(* Logix 5000 project; controller Arrow3 vendor 1 type 14 code 235 rev 36.11; software revision 36.00; part 2 of 3 *)
(* tags used below, declared in another part *)
   b : BOOL;
   off_delay_timer : TIMER;
   on : BOOL;
   On_Delay_Timer_1 : TIMER;
   On_Delay_Timer_2 : TIMER;
   On_Delay_Timer_3 : TIMER;
   On_Delay_Timer_4 : TIMER;
   On_Delay_Timer_5 : TIMER;
   On_Delay_Timer_6 : TIMER;
   On_Delay_Timer_7 : TIMER;
   On_Delay_Timer_8 : TIMER;
   on_delay_tmr : TIMER;
   PROP_BCKPLANE_IDENT_DEVICEID_GET : MESSAGE;
   PROP_BCKPLANE_IDENT_DEVICEID_TRG_GET : BOOL;
   PROP_BCKPLANE_IDENT_DEVICENAME_GET : MESSAGE;
   PROP_BCKPLANE_IDENT_DEVICENAME_TRG_GET : BOOL;
   PROP_BCKPLANE_IDENT_DEVICETYPE_GET : MESSAGE;
   PROP_BCKPLANE_IDENT_DEVICETYPE_TRG_GET : BOOL;
   PROP_BCKPLANE_IDENT_HWREV_GET : MESSAGE;
   PROP_BCKPLANE_IDENT_HWREV_TRG_GET : BOOL;
   PROP_BCKPLANE_IDENT_SERIALNO_GET : MESSAGE;
   PROP_BCKPLANE_IDENT_SERIALNO_TRG_GET : BOOL;
   PROP_BCKPLANE_IDENT_SWPARTNO_GET : MESSAGE;
   PROP_BCKPLANE_IDENT_SWPARTNO_TRG_GET : BOOL;
   PROP_BCKPLANE_IDENT_SWREV_GET : MESSAGE;
   PROP_BCKPLANE_IDENT_SWREV_TRG_GET : BOOL;
   PROP_BCKPLANE_IDENT_VARIANTID_GET : MESSAGE;
   PROP_BCKPLANE_IDENT_VARIANTID_TRG_GET : BOOL;
   PROP_BCKPLANE_IDENT_VENDORID_GET : MESSAGE;
   PROP_BCKPLANE_IDENT_VENDORID_TRG_GET : BOOL;
   PROP_BCKPLANE_IDENT_VENDORNAME_GET : MESSAGE;
   PROP_BCKPLANE_IDENT_VENDORNAME_TRG_GET : BOOL;
   PROP_INTR_CONTROL_KD_GET : MESSAGE;
   PROP_INTR_CONTROL_KD_SET : MESSAGE;
   PROP_INTR_CONTROL_KD_TRG_GET : BOOL;
   PROP_INTR_CONTROL_KD_TRG_SET : BOOL;
   PROP_INTR_CONTROL_KI_GET : MESSAGE;
   PROP_INTR_CONTROL_KI_SET : MESSAGE;
   PROP_INTR_CONTROL_KI_TRG_GET : BOOL;
   PROP_INTR_CONTROL_KI_TRG_SET : BOOL;
   PROP_INTR_CONTROL_KP_GET : MESSAGE;
   PROP_INTR_CONTROL_KP_SET : MESSAGE;
   PROP_INTR_CONTROL_KP_TRG_GET : BOOL;
   PROP_INTR_CONTROL_KP_TRG_SET : BOOL;
   PROP_INTR_CONTROL_LCDBRIGHT_GET : MESSAGE;
   PROP_INTR_CONTROL_LCDBRIGHT_SET : MESSAGE;
   PROP_INTR_CONTROL_LCDBRIGHT_TRG_GET : BOOL;
   PROP_INTR_CONTROL_LCDBRIGHT_TRG_SET : BOOL;
   PROP_INTR_CONTROL_SPANADJST_GET : MESSAGE;
   PROP_INTR_CONTROL_SPANADJST_SET : MESSAGE;
   PROP_INTR_CONTROL_SPANADJST_TRG_GET : BOOL;
   PROP_INTR_CONTROL_SPANADJST_TRG_SET : BOOL;
   PROP_INTR_CONTROL_ZEROADJST_GET : MESSAGE;
   PROP_INTR_CONTROL_ZEROADJST_SET : MESSAGE;
   PROP_INTR_CONTROL_ZEROADJST_TRG_GET : BOOL;
   PROP_INTR_CONTROL_ZEROADJST_TRG_SET : BOOL;
   PROP_INTR_CYCLECOUNTER_GET : MESSAGE;
   PROP_INTR_CYCLECOUNTER_TRG_GET : BOOL;
   PROP_INTR_IDENT_DEVICEID_GET : MESSAGE;
   PROP_INTR_IDENT_DEVICEID_TRG_GET : BOOL;
   PROP_INTR_IDENT_DEVICENAME_GET : MESSAGE;
   PROP_INTR_IDENT_DEVICENAME_TRG_GET : BOOL;
   PROP_INTR_IDENT_DEVICETYPE_GET : MESSAGE;
   PROP_INTR_IDENT_DEVICETYPE_TRG_GET : BOOL;
   PROP_INTR_IDENT_HWREV_GET : MESSAGE;
   PROP_INTR_IDENT_HWREV_TRG_GET : BOOL;
   PROP_INTR_IDENT_SERIALNO_GET : MESSAGE;
   PROP_INTR_IDENT_SERIALNO_TRG_GET : BOOL;
   PROP_INTR_IDENT_SWPARTNO_GET : MESSAGE;
   PROP_INTR_IDENT_SWPARTNO_TRG_GET : BOOL;
   PROP_INTR_IDENT_SWREV_GET : MESSAGE;
   PROP_INTR_IDENT_SWREV_TRG_GET : BOOL;
   PROP_INTR_IDENT_VARIANTID_GET : MESSAGE;
   PROP_INTR_IDENT_VARIANTID_TRG_GET : BOOL;
   PROP_INTR_IDENT_VENDORID_GET : MESSAGE;
   PROP_INTR_IDENT_VENDORID_TRG_GET : BOOL;
   PROP_INTR_IDENT_VENDORNAME_GET : MESSAGE;
   PROP_INTR_IDENT_VENDORNAME_TRG_GET : BOOL;
   PROP_INTR_OPRHR_GET : MESSAGE;
   PROP_INTR_OPRHR_TRG_GET : BOOL;
   PROP_INTR_POST_ERRSTS_GET : MESSAGE;
   PROP_INTR_POST_ERRSTS_TRG_GET : BOOL;
   STA_ApplPresHysteresis_GET : MESSAGE;
   STA_ApplPresHysteresis_SET : MESSAGE;
   STA_ApplPresHysteresis_TRG_GET : BOOL;
   STA_ApplPresHysteresis_TRG_SET : BOOL;
   STA_Coil12HitCurHysteresis_GET : MESSAGE;
   STA_Coil12HitCurHysteresis_SET : MESSAGE;
   STA_Coil12HitCurHysteresis_TRG_GET : BOOL;
   STA_Coil12HitCurHysteresis_TRG_SET : BOOL;
   STA_Coil12HitCurrent_GET : MESSAGE;
   STA_Coil12HitCurrent_TRG_GET : BOOL;
   STA_Coil12HitPower_GET : MESSAGE;
   STA_Coil12HitPower_TRG_GET : BOOL;
   STA_Coil12HoldCurrent_GET : MESSAGE;
   STA_Coil12HoldCurrent_TRG_GET : BOOL;
   STA_Coil12HoldPower_GET : MESSAGE;
   STA_Coil12HoldPower_SET : MESSAGE;
   STA_Coil12HoldPower_TRG_GET : BOOL;
   STA_Coil12HoldPower_TRG_SET : BOOL;
   STA_Coil12HoldVolage_GET : MESSAGE;
   STA_Coil12HoldVolage_SET : MESSAGE;
   STA_Coil12HoldVolage_TRG_GET : BOOL;
   STA_Coil12HoldVolage_TRG_SET : BOOL;
   STA_Coil14HitCurHysteresis_GET : MESSAGE;
   STA_Coil14HitCurHysteresis_SET : MESSAGE;
   STA_Coil14HitCurHysteresis_TRG_GET : BOOL;
   STA_Coil14HitCurHysteresis_TRG_SET : BOOL;
   STA_Coil14HitCurrent_GET : MESSAGE;
   STA_Coil14HitCurrent_TRG_GET : BOOL;
   STA_Coil14HitPower_GET : MESSAGE;
   STA_Coil14HitPower_TRG_GET : BOOL;
   STA_Coil14HoldCurrent_GET : MESSAGE;
   STA_Coil14HoldCurrent_TRG_GET : BOOL;
   STA_Coil14HoldPower_GET : MESSAGE;
   STA_Coil14HoldPower_SET : MESSAGE;
   STA_Coil14HoldPower_TRG_GET : BOOL;
   STA_Coil14HoldPower_TRG_SET : BOOL;
   STA_Coil14HoldVolage_GET : MESSAGE;
   STA_Coil14HoldVolage_SET : MESSAGE;
   STA_Coil14HoldVolage_TRG_GET : BOOL;
   STA_Coil14HoldVolage_TRG_SET : BOOL;
   STA_DV_ERROR_STATUS_GET : MESSAGE;
   STA_DV_ERROR_STATUS_TRG_GET : BOOL;
   STA_ExhaustPresHysteresis_GET : MESSAGE;
   STA_ExhaustPresHysteresis_SET : MESSAGE;
   STA_ExhaustPresHysteresis_TRG_GET : BOOL;
   STA_ExhaustPresHysteresis_TRG_SET : BOOL;
   STA_FAULTEVNTBITS_GET : MESSAGE;
   STA_FAULTEVNTBITS_TRG_GET : BOOL;
   STA_FAULTEVNTCOUNT_GET : MESSAGE;
   STA_FAULTEVNTCOUNT_TRG_GET : BOOL;
   STA_IDENT_DEVICETYPE_GET : MESSAGE;
   STA_IDENT_DEVICETYPE_TRG_GET : BOOL;
   STA_INTR_IDENT_DEVICEID_GET : MESSAGE;
   STA_INTR_IDENT_DEVICEID_TRG_GET : BOOL;
   STA_INTR_IDENT_DEVICENAME_GET : MESSAGE;
   STA_INTR_IDENT_DEVICENAME_TRG_GET : BOOL;
   STA_INTR_IDENT_HWREV_GET : MESSAGE;
   STA_INTR_IDENT_HWREV_TRG_GET : BOOL;
   STA_INTR_IDENT_SERIALNO_GET : MESSAGE;
   STA_INTR_IDENT_SERIALNO_TRG_GET : BOOL;
   STA_INTR_IDENT_SWPARTNO_GET : MESSAGE;
   STA_INTR_IDENT_SWPARTNO_TRG_GET : BOOL;
   STA_INTR_IDENT_SWREV_GET : MESSAGE;
   STA_INTR_IDENT_SWREV_TRG_GET : BOOL;
   STA_INTR_IDENT_VARIANTID_GET : MESSAGE;
   STA_INTR_IDENT_VARIANTID_TRG_GET : BOOL;
   STA_INTR_IDENT_VENDORID_GET : MESSAGE;
   STA_INTR_IDENT_VENDORID_TRG_GET : BOOL;
   STA_INTR_IDENT_VENDORNAME_GET : MESSAGE;
   STA_INTR_IDENT_VENDORNAME_TRG_GET : BOOL;
   STA_MaxApplPressure_GET : MESSAGE;
   STA_MaxApplPressure_SET : MESSAGE;
   STA_MaxApplPressure_TRG_GET : BOOL;
   STA_MaxApplPressure_TRG_SET : BOOL;
   STA_MeasuredAuxVolt_GET : MESSAGE;
   STA_MeasuredAuxVolt_TRG_GET : BOOL;
   STA_MinApplPressure_GET : MESSAGE;
   STA_MinApplPressure_SET : MESSAGE;
   STA_MinApplPressure_TRG_GET : BOOL;
   STA_MinApplPressure_TRG_SET : BOOL;
   STA_OPERATIONTIME_HR_GET : MESSAGE;
   STA_OPERATIONTIME_HR_TRG_GET : BOOL;
   STA_OPERATIONTIME_MIN_GET : MESSAGE;
   STA_OPERATIONTIME_MIN_TRG_GET : BOOL;
   STA_Port2ApplPressCyclRating_GET : MESSAGE;
   STA_Port2ApplPressCyclRating_SET : MESSAGE;
   STA_Port2ApplPressCyclRating_TRG_GET : BOOL;
   STA_Port2ApplPressCyclRating_TRG_SET : BOOL;
   STA_Port2MesrdPressure_GET : MESSAGE;
   STA_Port2MesrdPressure_TRG_GET : BOOL;
   STA_Port2PressCycleCounter_GET : MESSAGE;
   STA_Port2PressCycleCounter_TRG_GET : BOOL;
   STA_Port2PressMonitorDly_GET : MESSAGE;
   STA_Port2PressMonitorDly_SET : MESSAGE;
   STA_Port2PressMonitorDly_TRG_GET : BOOL;
   STA_Port2PressMonitorDly_TRG_SET : BOOL;
   STA_Port4ApplPressCyclRating_GET : MESSAGE;
   STA_Port4ApplPressCyclRating_SET : MESSAGE;
   STA_Port4ApplPressCyclRating_TRG_GET : BOOL;
   STA_Port4ApplPressCyclRating_TRG_SET : BOOL;
   STA_Port4MesrdPressure_GET : MESSAGE;
   STA_Port4MesrdPressure_TRG_GET : BOOL;
   STA_Port4PressCycleCounter_GET : MESSAGE;
   STA_Port4PressCycleCounter_TRG_GET : BOOL;
   STA_Port4PressMonitorDly_GET : MESSAGE;
   STA_Port4PressMonitorDly_SET : MESSAGE;
   STA_Port4PressMonitorDly_TRG_GET : BOOL;
   STA_Port4PressMonitorDly_TRG_SET : BOOL;
   STA_PWRONTIME_HR_GET : MESSAGE;
   STA_PWRONTIME_HR_TRG_GET : BOOL;
   STA_PWRONTIME_MIN_GET : MESSAGE;
   STA_PWRONTIME_MIN_TRG_GET : BOOL;
   STA_RatedAuxVoltHyst_GET : MESSAGE;
   STA_RatedAuxVoltHyst_SET : MESSAGE;
   STA_RatedAuxVoltHyst_TRG_GET : BOOL;
   STA_RatedAuxVoltHyst_TRG_SET : BOOL;
   STA_Valve12ApplCyclRating_GET : MESSAGE;
   STA_Valve12ApplCyclRating_SET : MESSAGE;
   STA_Valve12ApplCyclRating_TRG_GET : BOOL;
   STA_Valve12ApplCyclRating_TRG_SET : BOOL;
   STA_Valve12CycleCounter_GET : MESSAGE;
   STA_Valve12CycleCounter_TRG_GET : BOOL;
   STA_Valve14ApplCyclRating_GET : MESSAGE;
   STA_Valve14ApplCyclRating_SET : MESSAGE;
   STA_Valve14ApplCyclRating_TRG_GET : BOOL;
   STA_Valve14ApplCyclRating_TRG_SET : BOOL;
   STA_Valve14CycleCounter_GET : MESSAGE;
   STA_Valve14CycleCounter_TRG_GET : BOOL;
   STA_ValveSlice12Side_GET : MESSAGE;
   STA_ValveSlice12Side_SET : MESSAGE;
   STA_ValveSlice12Side_TRG_GET : BOOL;
   STA_ValveSlice12Side_TRG_SET : BOOL;
   STA_ValveSliceFunction_GET : MESSAGE;
   STA_ValveSliceFunction_SET : MESSAGE;
   STA_ValveSliceFunction_TRG_GET : BOOL;
   STA_ValveSliceFunction_TRG_SET : BOOL;
   STA_WARNEVNTBITS_GET : MESSAGE;
   STA_WARNEVNTBITS_TRG_GET : BOOL;
   STA_WARNEVNTCOUNT_GET : MESSAGE;
   STA_WARNEVNTCOUNT_TRG_GET : BOOL;
   STA_WARNSTSBITS_GET : MESSAGE;
   STA_WARNSTSBITS_TRG_GET : BOOL;
   Station_1A : ALIAS FOR VRQx:O.Data[1].7;
   Station_1B : ALIAS FOR VRQx:O.Data[1].6;
   Station_2A : ALIAS FOR VRQx:O.Data[1].5;
   Station_2B : ALIAS FOR VRQx:O.Data[1].4;
   Station_3A : ALIAS FOR VRQx:O.Data[1].3;
   Station_3B : ALIAS FOR VRQx:O.Data[1].2;
   Station_4A : ALIAS FOR VRQx:O.Data[1].1;
   Station_4B : ALIAS FOR VRQx:O.Data[1].0;
   Station_5A : ALIAS FOR VRQx:O.Data[2].7;
   Station_5B : ALIAS FOR VRQx:O.Data[2].6;
   Station_6A : ALIAS FOR VRQx:O.Data[2].5;
   Station_6B : ALIAS FOR VRQx:O.Data[2].4;
   Station_7A : ALIAS FOR VRQx:O.Data[2].3;
   Station_7B : ALIAS FOR VRQx:O.Data[2].2;
   Station_8A : ALIAS FOR VRQx:O.Data[2].1;
   Station_8B : ALIAS FOR VRQx:O.Data[2].0;
   up_counter : COUNTER;
(* MainProgram, continued *)

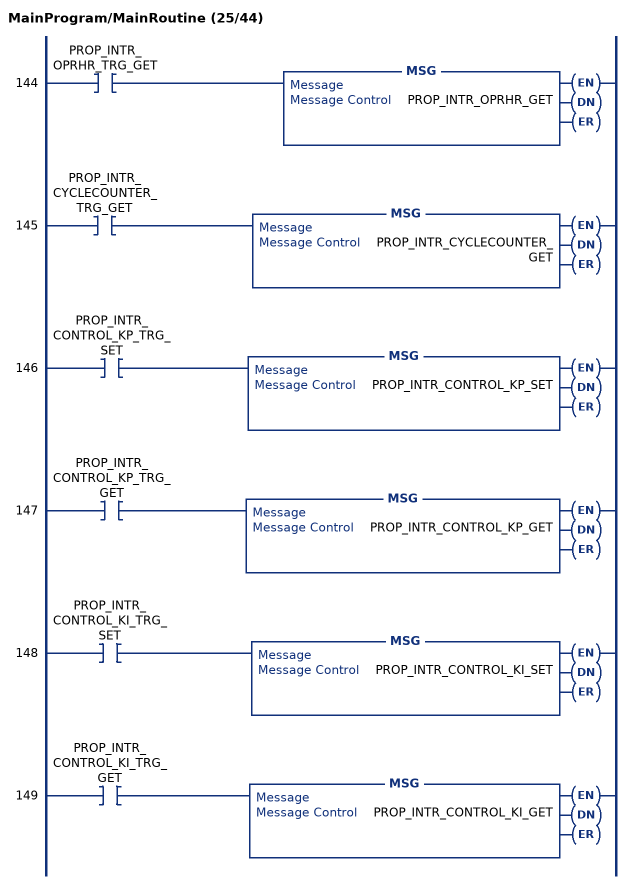
   [picture p24: MainProgram/MainRoutine rungs 144-149]
   144: XIC(PROP_INTR_OPRHR_TRG_GET)MSG(PROP_INTR_OPRHR_GET);
   145: XIC(PROP_INTR_CYCLECOUNTER_TRG_GET)MSG(PROP_INTR_CYCLECOUNTER_GET);
   146: XIC(PROP_INTR_CONTROL_KP_TRG_SET)MSG(PROP_INTR_CONTROL_KP_SET);
   147: XIC(PROP_INTR_CONTROL_KP_TRG_GET)MSG(PROP_INTR_CONTROL_KP_GET);
   148: XIC(PROP_INTR_CONTROL_KI_TRG_SET)MSG(PROP_INTR_CONTROL_KI_SET);
   149: XIC(PROP_INTR_CONTROL_KI_TRG_GET)MSG(PROP_INTR_CONTROL_KI_GET);
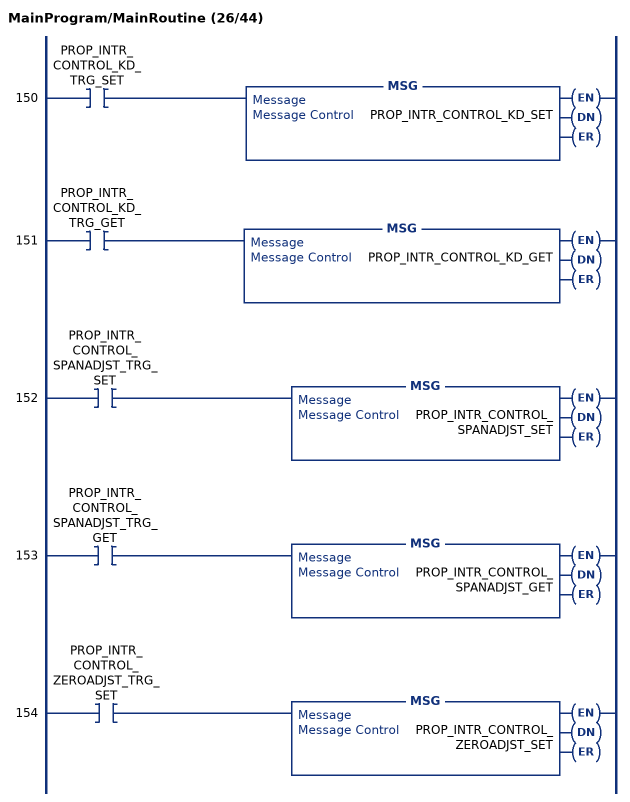
   150: XIC(PROP_INTR_CONTROL_KD_TRG_SET)MSG(PROP_INTR_CONTROL_KD_SET);
   151: XIC(PROP_INTR_CONTROL_KD_TRG_GET)MSG(PROP_INTR_CONTROL_KD_GET);
   152: XIC(PROP_INTR_CONTROL_SPANADJST_TRG_SET)MSG(PROP_INTR_CONTROL_SPANADJST_SET);
   153: XIC(PROP_INTR_CONTROL_SPANADJST_TRG_GET)MSG(PROP_INTR_CONTROL_SPANADJST_GET);
   154: XIC(PROP_INTR_CONTROL_ZEROADJST_TRG_SET)MSG(PROP_INTR_CONTROL_ZEROADJST_SET);
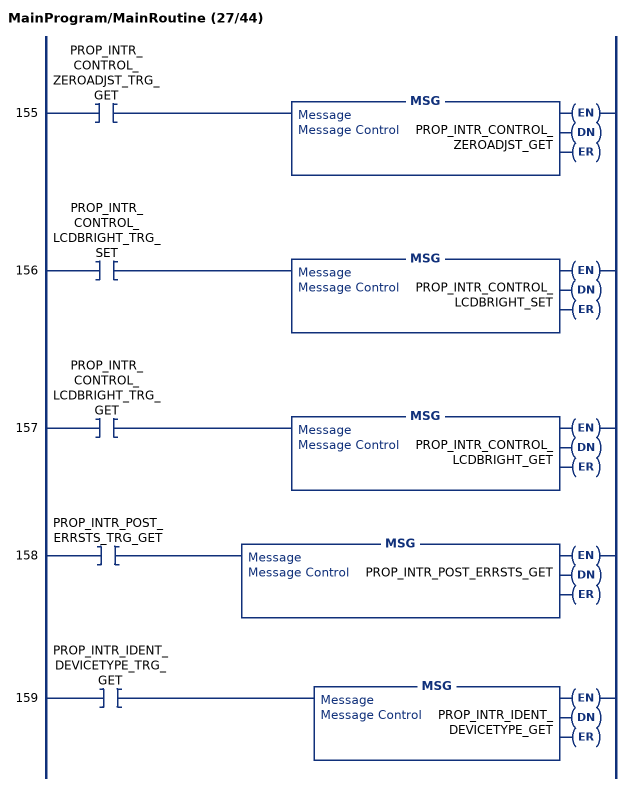
   155: XIC(PROP_INTR_CONTROL_ZEROADJST_TRG_GET)MSG(PROP_INTR_CONTROL_ZEROADJST_GET);
   156: XIC(PROP_INTR_CONTROL_LCDBRIGHT_TRG_SET)MSG(PROP_INTR_CONTROL_LCDBRIGHT_SET);
   157: XIC(PROP_INTR_CONTROL_LCDBRIGHT_TRG_GET)MSG(PROP_INTR_CONTROL_LCDBRIGHT_GET);
   158: XIC(PROP_INTR_POST_ERRSTS_TRG_GET)MSG(PROP_INTR_POST_ERRSTS_GET);
   159: XIC(PROP_INTR_IDENT_DEVICETYPE_TRG_GET)MSG(PROP_INTR_IDENT_DEVICETYPE_GET);
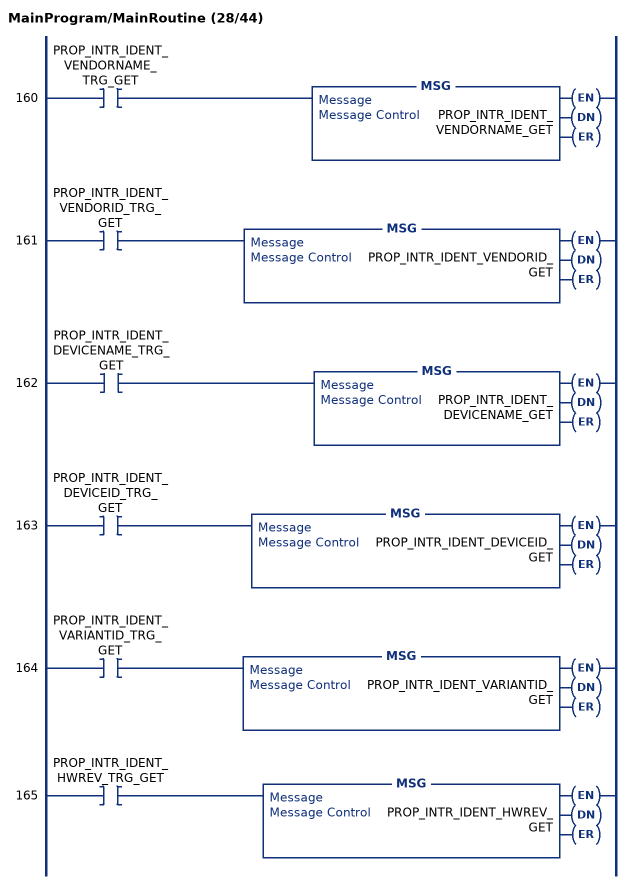
   160: XIC(PROP_INTR_IDENT_VENDORNAME_TRG_GET)MSG(PROP_INTR_IDENT_VENDORNAME_GET);
   161: XIC(PROP_INTR_IDENT_VENDORID_TRG_GET)MSG(PROP_INTR_IDENT_VENDORID_GET);
   162: XIC(PROP_INTR_IDENT_DEVICENAME_TRG_GET)MSG(PROP_INTR_IDENT_DEVICENAME_GET);
   163: XIC(PROP_INTR_IDENT_DEVICEID_TRG_GET)MSG(PROP_INTR_IDENT_DEVICEID_GET);
   164: XIC(PROP_INTR_IDENT_VARIANTID_TRG_GET)MSG(PROP_INTR_IDENT_VARIANTID_GET);
   165: XIC(PROP_INTR_IDENT_HWREV_TRG_GET)MSG(PROP_INTR_IDENT_HWREV_GET);
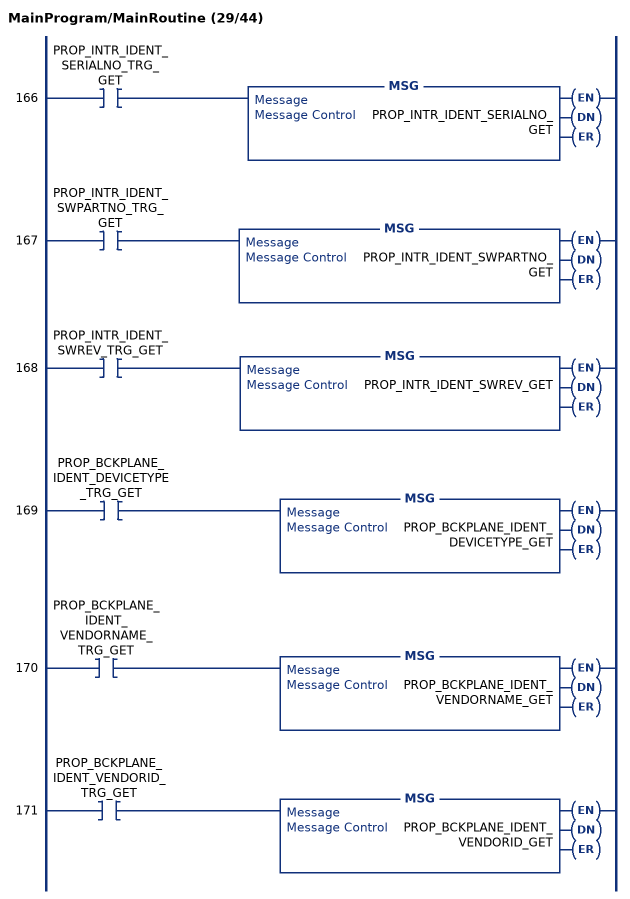
   166: XIC(PROP_INTR_IDENT_SERIALNO_TRG_GET)MSG(PROP_INTR_IDENT_SERIALNO_GET);
   167: XIC(PROP_INTR_IDENT_SWPARTNO_TRG_GET)MSG(PROP_INTR_IDENT_SWPARTNO_GET);
   168: XIC(PROP_INTR_IDENT_SWREV_TRG_GET)MSG(PROP_INTR_IDENT_SWREV_GET);
   169: XIC(PROP_BCKPLANE_IDENT_DEVICETYPE_TRG_GET)MSG(PROP_BCKPLANE_IDENT_DEVICETYPE_GET);
   170: XIC(PROP_BCKPLANE_IDENT_VENDORNAME_TRG_GET)MSG(PROP_BCKPLANE_IDENT_VENDORNAME_GET);
   171: XIC(PROP_BCKPLANE_IDENT_VENDORID_TRG_GET)MSG(PROP_BCKPLANE_IDENT_VENDORID_GET);
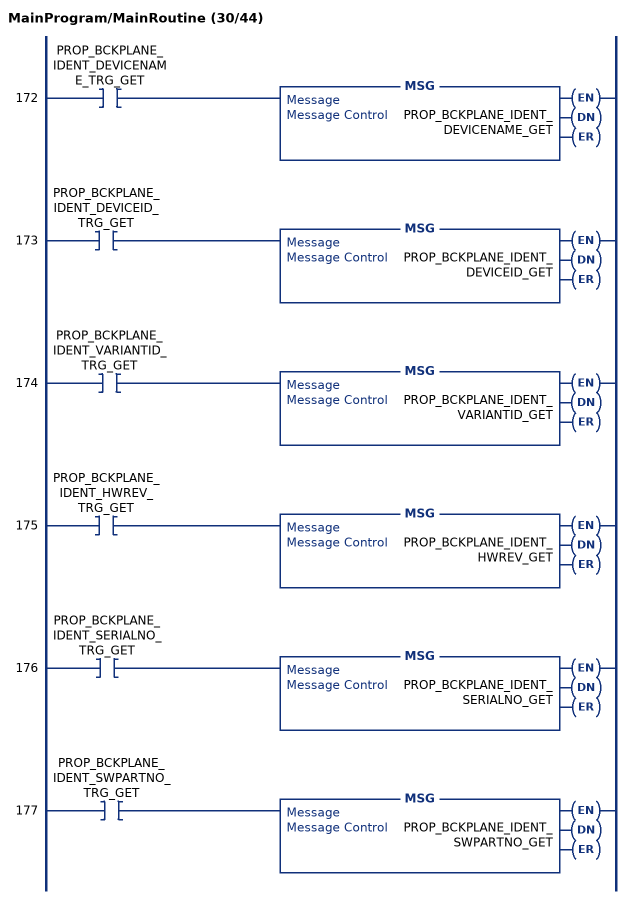
   172: XIC(PROP_BCKPLANE_IDENT_DEVICENAME_TRG_GET)MSG(PROP_BCKPLANE_IDENT_DEVICENAME_GET);
   173: XIC(PROP_BCKPLANE_IDENT_DEVICEID_TRG_GET)MSG(PROP_BCKPLANE_IDENT_DEVICEID_GET);
   174: XIC(PROP_BCKPLANE_IDENT_VARIANTID_TRG_GET)MSG(PROP_BCKPLANE_IDENT_VARIANTID_GET);
   175: XIC(PROP_BCKPLANE_IDENT_HWREV_TRG_GET)MSG(PROP_BCKPLANE_IDENT_HWREV_GET);
   176: XIC(PROP_BCKPLANE_IDENT_SERIALNO_TRG_GET)MSG(PROP_BCKPLANE_IDENT_SERIALNO_GET);
   177: XIC(PROP_BCKPLANE_IDENT_SWPARTNO_TRG_GET)MSG(PROP_BCKPLANE_IDENT_SWPARTNO_GET);
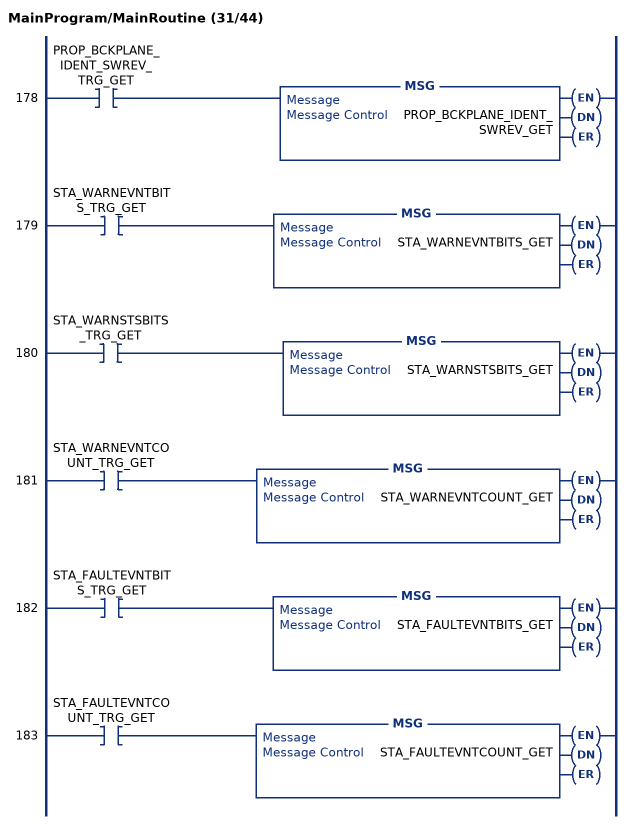
   178: XIC(PROP_BCKPLANE_IDENT_SWREV_TRG_GET)MSG(PROP_BCKPLANE_IDENT_SWREV_GET);
   179: XIC(STA_WARNEVNTBITS_TRG_GET)MSG(STA_WARNEVNTBITS_GET);
   180: XIC(STA_WARNSTSBITS_TRG_GET)MSG(STA_WARNSTSBITS_GET);
   181: XIC(STA_WARNEVNTCOUNT_TRG_GET)MSG(STA_WARNEVNTCOUNT_GET);
   182: XIC(STA_FAULTEVNTBITS_TRG_GET)MSG(STA_FAULTEVNTBITS_GET);
   183: XIC(STA_FAULTEVNTCOUNT_TRG_GET)MSG(STA_FAULTEVNTCOUNT_GET);
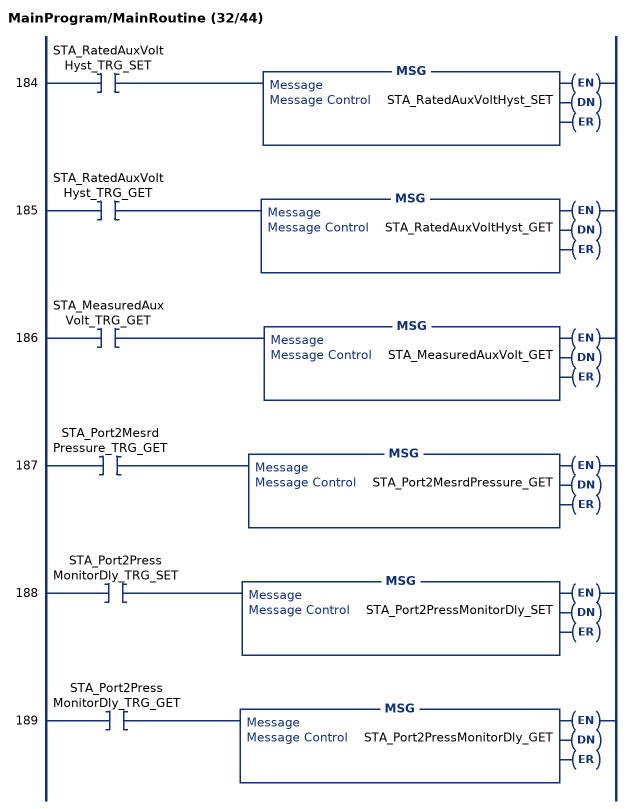
   184: XIC(STA_RatedAuxVoltHyst_TRG_SET)MSG(STA_RatedAuxVoltHyst_SET);
   185: XIC(STA_RatedAuxVoltHyst_TRG_GET)MSG(STA_RatedAuxVoltHyst_GET);
   186: XIC(STA_MeasuredAuxVolt_TRG_GET)MSG(STA_MeasuredAuxVolt_GET);
   187: XIC(STA_Port2MesrdPressure_TRG_GET)MSG(STA_Port2MesrdPressure_GET);
   188: XIC(STA_Port2PressMonitorDly_TRG_SET)MSG(STA_Port2PressMonitorDly_SET);
   189: XIC(STA_Port2PressMonitorDly_TRG_GET)MSG(STA_Port2PressMonitorDly_GET);
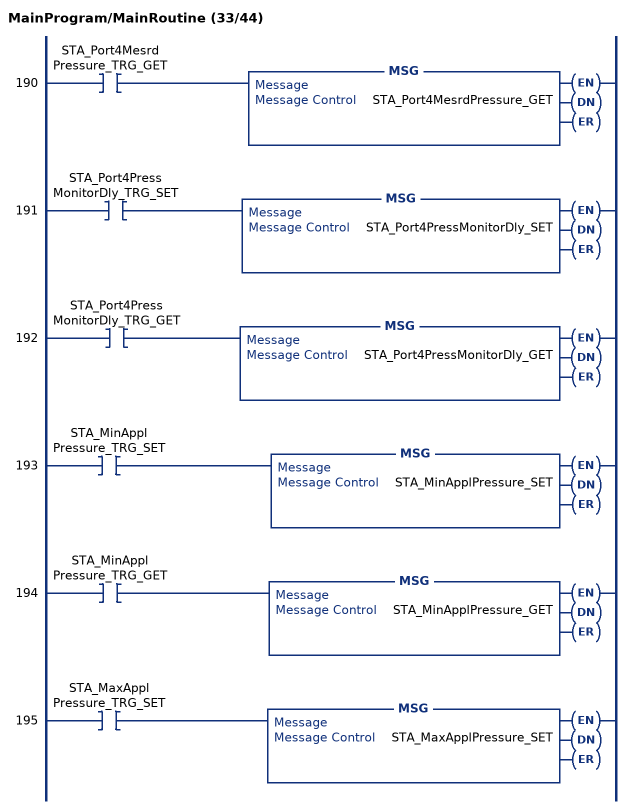
   190: XIC(STA_Port4MesrdPressure_TRG_GET)MSG(STA_Port4MesrdPressure_GET);
   191: XIC(STA_Port4PressMonitorDly_TRG_SET)MSG(STA_Port4PressMonitorDly_SET);
   192: XIC(STA_Port4PressMonitorDly_TRG_GET)MSG(STA_Port4PressMonitorDly_GET);
   193: XIC(STA_MinApplPressure_TRG_SET)MSG(STA_MinApplPressure_SET);
   194: XIC(STA_MinApplPressure_TRG_GET)MSG(STA_MinApplPressure_GET);
   195: XIC(STA_MaxApplPressure_TRG_SET)MSG(STA_MaxApplPressure_SET);
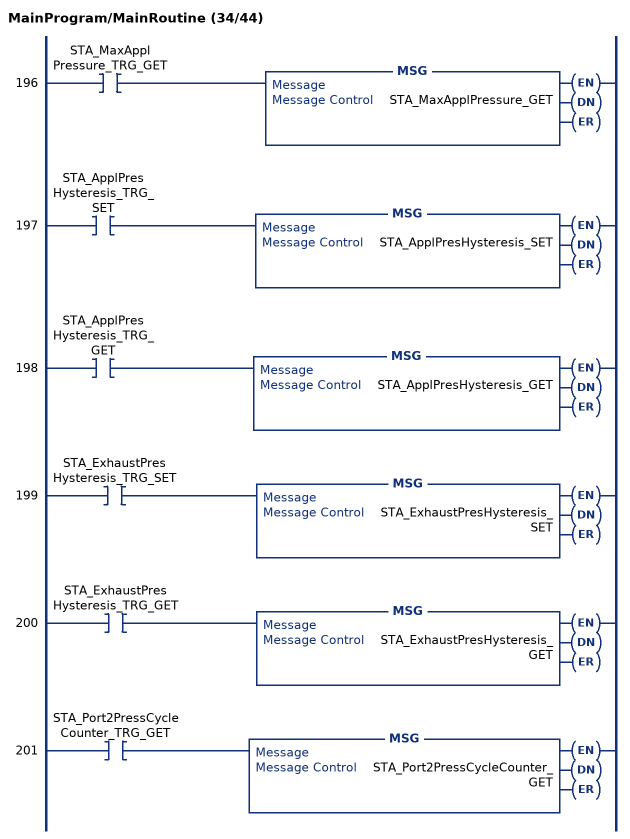
   196: XIC(STA_MaxApplPressure_TRG_GET)MSG(STA_MaxApplPressure_GET);
   197: XIC(STA_ApplPresHysteresis_TRG_SET)MSG(STA_ApplPresHysteresis_SET);
   198: XIC(STA_ApplPresHysteresis_TRG_GET)MSG(STA_ApplPresHysteresis_GET);
   199: XIC(STA_ExhaustPresHysteresis_TRG_SET)MSG(STA_ExhaustPresHysteresis_SET);
   200: XIC(STA_ExhaustPresHysteresis_TRG_GET)MSG(STA_ExhaustPresHysteresis_GET);
   201: XIC(STA_Port2PressCycleCounter_TRG_GET)MSG(STA_Port2PressCycleCounter_GET);
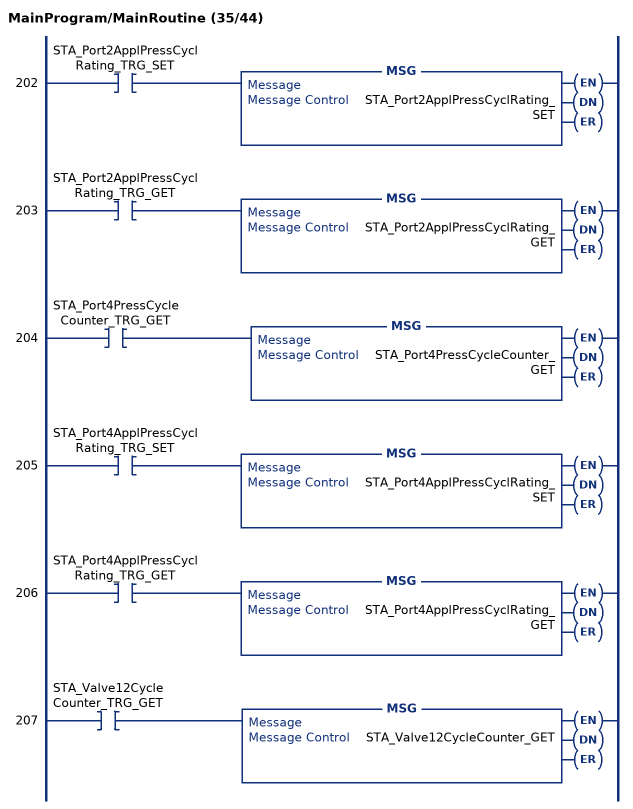
   202: XIC(STA_Port2ApplPressCyclRating_TRG_SET)MSG(STA_Port2ApplPressCyclRating_SET);
   203: XIC(STA_Port2ApplPressCyclRating_TRG_GET)MSG(STA_Port2ApplPressCyclRating_GET);
   204: XIC(STA_Port4PressCycleCounter_TRG_GET)MSG(STA_Port4PressCycleCounter_GET);
   205: XIC(STA_Port4ApplPressCyclRating_TRG_SET)MSG(STA_Port4ApplPressCyclRating_SET);
   206: XIC(STA_Port4ApplPressCyclRating_TRG_GET)MSG(STA_Port4ApplPressCyclRating_GET);
   207: XIC(STA_Valve12CycleCounter_TRG_GET)MSG(STA_Valve12CycleCounter_GET);
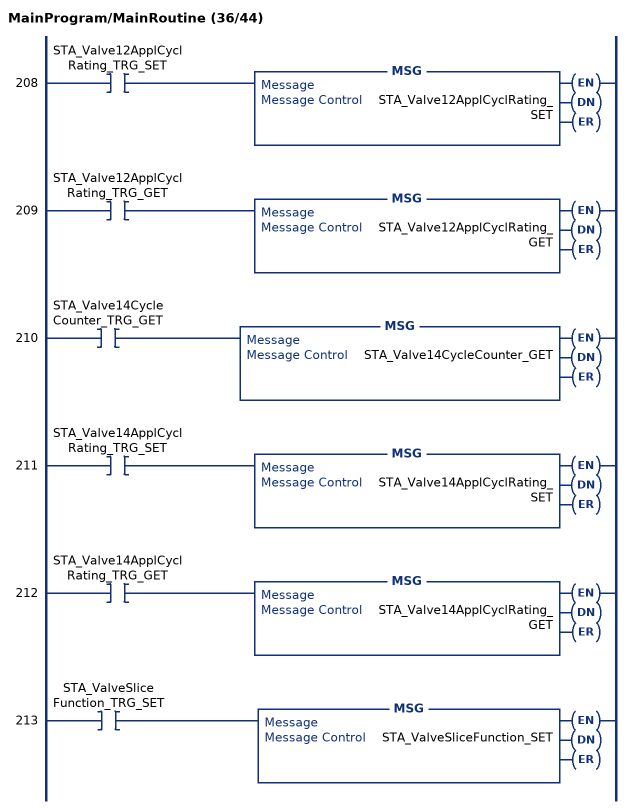
   208: XIC(STA_Valve12ApplCyclRating_TRG_SET)MSG(STA_Valve12ApplCyclRating_SET);
   209: XIC(STA_Valve12ApplCyclRating_TRG_GET)MSG(STA_Valve12ApplCyclRating_GET);
   210: XIC(STA_Valve14CycleCounter_TRG_GET)MSG(STA_Valve14CycleCounter_GET);
   211: XIC(STA_Valve14ApplCyclRating_TRG_SET)MSG(STA_Valve14ApplCyclRating_SET);
   212: XIC(STA_Valve14ApplCyclRating_TRG_GET)MSG(STA_Valve14ApplCyclRating_GET);
   213: XIC(STA_ValveSliceFunction_TRG_SET)MSG(STA_ValveSliceFunction_SET);
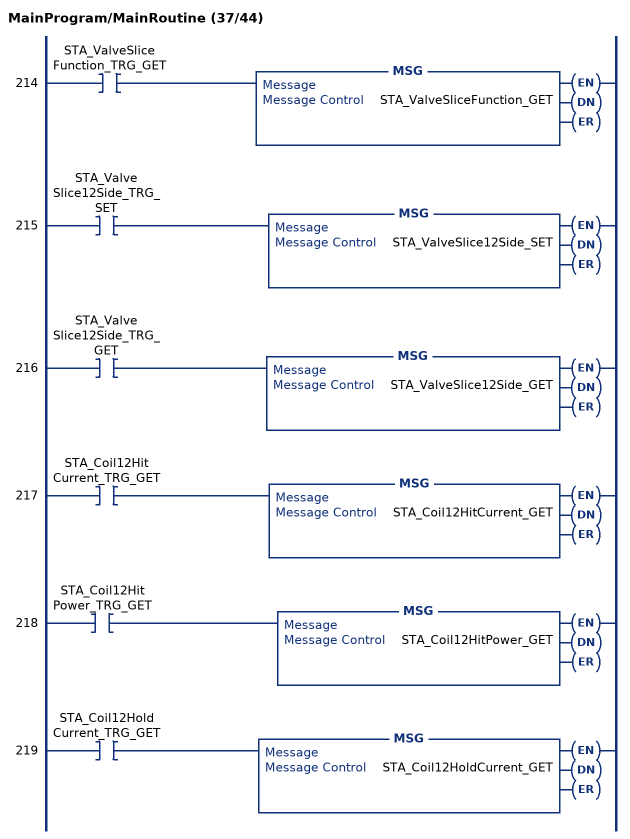
   214: XIC(STA_ValveSliceFunction_TRG_GET)MSG(STA_ValveSliceFunction_GET);
   215: XIC(STA_ValveSlice12Side_TRG_SET)MSG(STA_ValveSlice12Side_SET);
   216: XIC(STA_ValveSlice12Side_TRG_GET)MSG(STA_ValveSlice12Side_GET);
   217: XIC(STA_Coil12HitCurrent_TRG_GET)MSG(STA_Coil12HitCurrent_GET);
   218: XIC(STA_Coil12HitPower_TRG_GET)MSG(STA_Coil12HitPower_GET);
   219: XIC(STA_Coil12HoldCurrent_TRG_GET)MSG(STA_Coil12HoldCurrent_GET);
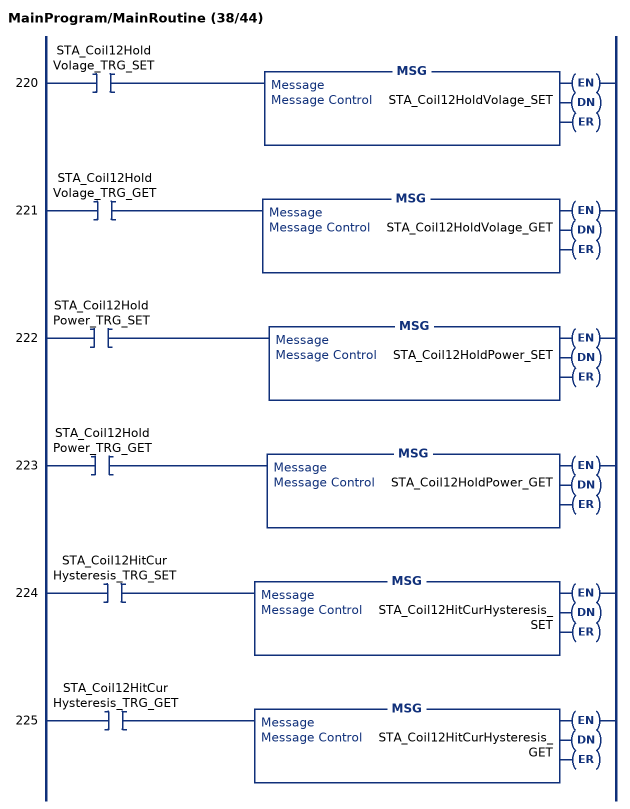
   220: XIC(STA_Coil12HoldVolage_TRG_SET)MSG(STA_Coil12HoldVolage_SET);
   221: XIC(STA_Coil12HoldVolage_TRG_GET)MSG(STA_Coil12HoldVolage_GET);
   222: XIC(STA_Coil12HoldPower_TRG_SET)MSG(STA_Coil12HoldPower_SET);
   223: XIC(STA_Coil12HoldPower_TRG_GET)MSG(STA_Coil12HoldPower_GET);
   224: XIC(STA_Coil12HitCurHysteresis_TRG_SET)MSG(STA_Coil12HitCurHysteresis_SET);
   225: XIC(STA_Coil12HitCurHysteresis_TRG_GET)MSG(STA_Coil12HitCurHysteresis_GET);
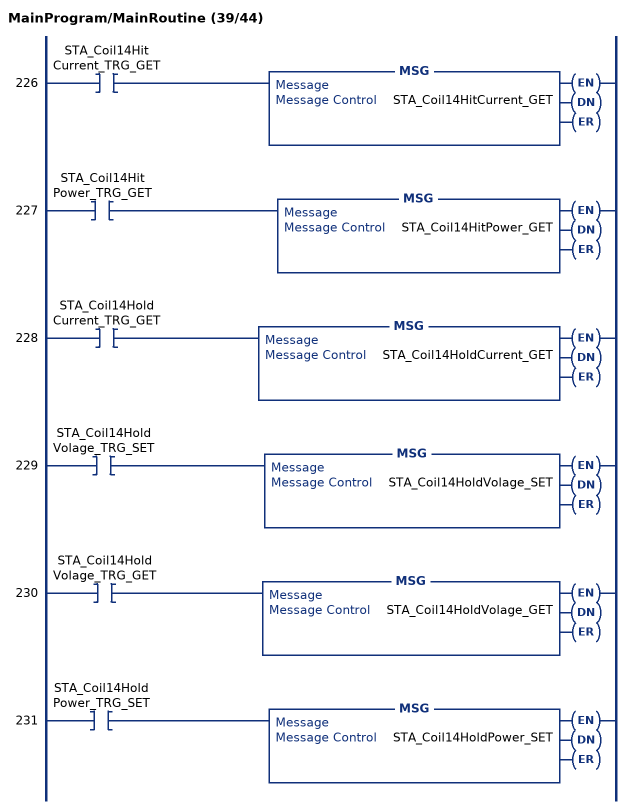
   226: XIC(STA_Coil14HitCurrent_TRG_GET)MSG(STA_Coil14HitCurrent_GET);
   227: XIC(STA_Coil14HitPower_TRG_GET)MSG(STA_Coil14HitPower_GET);
   228: XIC(STA_Coil14HoldCurrent_TRG_GET)MSG(STA_Coil14HoldCurrent_GET);
   229: XIC(STA_Coil14HoldVolage_TRG_SET)MSG(STA_Coil14HoldVolage_SET);
   230: XIC(STA_Coil14HoldVolage_TRG_GET)MSG(STA_Coil14HoldVolage_GET);
   231: XIC(STA_Coil14HoldPower_TRG_SET)MSG(STA_Coil14HoldPower_SET);
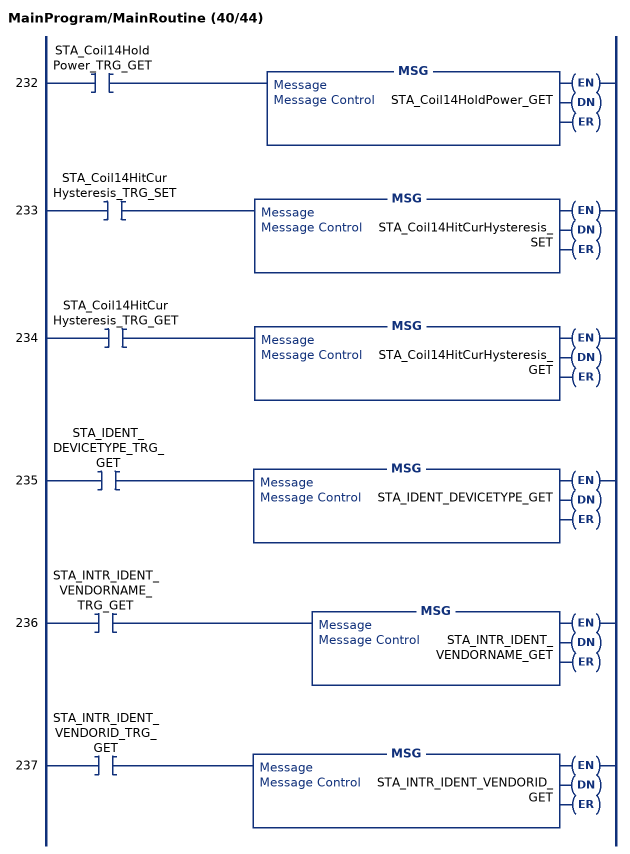
   232: XIC(STA_Coil14HoldPower_TRG_GET)MSG(STA_Coil14HoldPower_GET);
   233: XIC(STA_Coil14HitCurHysteresis_TRG_SET)MSG(STA_Coil14HitCurHysteresis_SET);
   234: XIC(STA_Coil14HitCurHysteresis_TRG_GET)MSG(STA_Coil14HitCurHysteresis_GET);
   235: XIC(STA_IDENT_DEVICETYPE_TRG_GET)MSG(STA_IDENT_DEVICETYPE_GET);
   236: XIC(STA_INTR_IDENT_VENDORNAME_TRG_GET)MSG(STA_INTR_IDENT_VENDORNAME_GET);
   237: XIC(STA_INTR_IDENT_VENDORID_TRG_GET)MSG(STA_INTR_IDENT_VENDORID_GET);
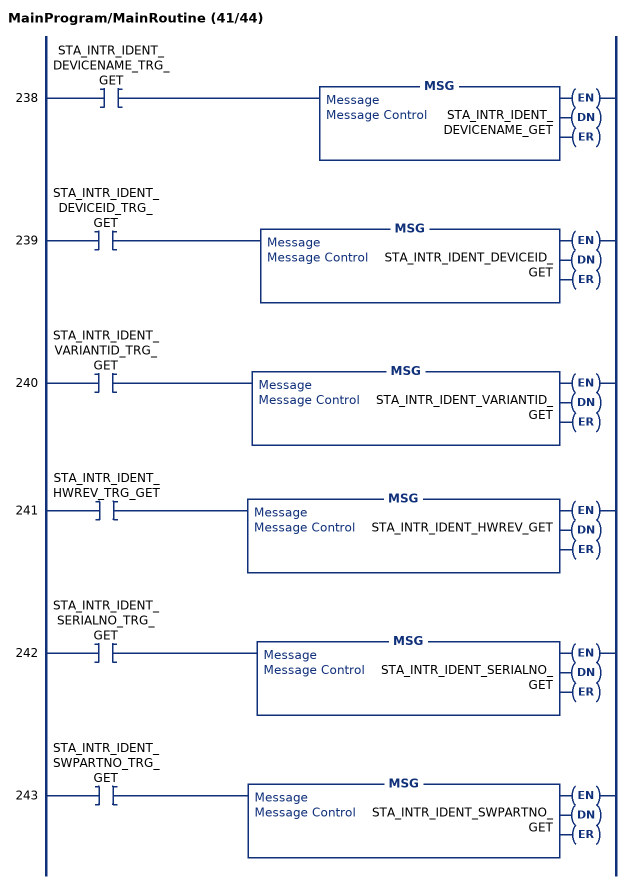
   238: XIC(STA_INTR_IDENT_DEVICENAME_TRG_GET)MSG(STA_INTR_IDENT_DEVICENAME_GET);
   239: XIC(STA_INTR_IDENT_DEVICEID_TRG_GET)MSG(STA_INTR_IDENT_DEVICEID_GET);
   240: XIC(STA_INTR_IDENT_VARIANTID_TRG_GET)MSG(STA_INTR_IDENT_VARIANTID_GET);
   241: XIC(STA_INTR_IDENT_HWREV_TRG_GET)MSG(STA_INTR_IDENT_HWREV_GET);
   242: XIC(STA_INTR_IDENT_SERIALNO_TRG_GET)MSG(STA_INTR_IDENT_SERIALNO_GET);
   243: XIC(STA_INTR_IDENT_SWPARTNO_TRG_GET)MSG(STA_INTR_IDENT_SWPARTNO_GET);
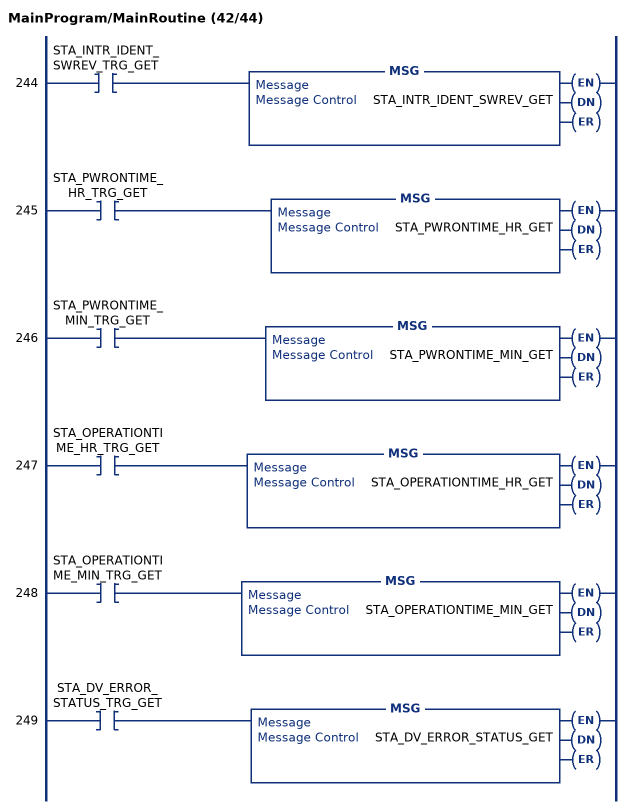
   244: XIC(STA_INTR_IDENT_SWREV_TRG_GET)MSG(STA_INTR_IDENT_SWREV_GET);
   245: XIC(STA_PWRONTIME_HR_TRG_GET)MSG(STA_PWRONTIME_HR_GET);
   246: XIC(STA_PWRONTIME_MIN_TRG_GET)MSG(STA_PWRONTIME_MIN_GET);
   247: XIC(STA_OPERATIONTIME_HR_TRG_GET)MSG(STA_OPERATIONTIME_HR_GET);
   248: XIC(STA_OPERATIONTIME_MIN_TRG_GET)MSG(STA_OPERATIONTIME_MIN_GET);
   249: XIC(STA_DV_ERROR_STATUS_TRG_GET)MSG(STA_DV_ERROR_STATUS_GET);
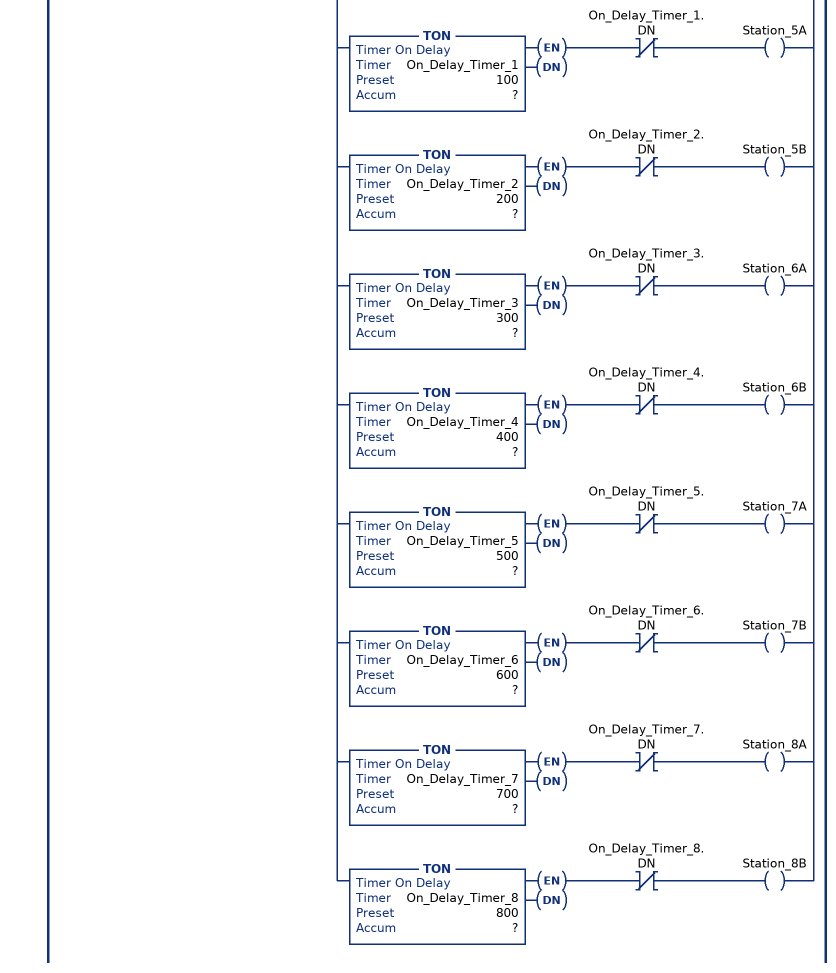
   250: XIC(on)CTU(up_counter,?,?)[TON(On_Delay_Timer_1,?,?) XIO(On_Delay_Timer_1.DN) OTE(Station_1A) ,TON(On_Delay_Timer_2,?,?) XIO(On_Delay_Timer_2.DN) OTE(Station_1B) ,TON(On_Delay_Timer_3,?,?) XIO(On_Delay_Timer_3.DN) OTE(Station_2A) ,TON(On_Delay_Timer_4,?,?) XIO(On_Delay_Timer_4.DN) OTE(Station_2B) ,TON(On_Delay_Timer_5,?,?) XIO(On_Delay_Timer_5.DN) OTE(Station_3A) ,TON(On_Delay_Timer_6,?,?) XIO(On_Delay_Timer_6.DN) OTE(Station_3B) ,TON(On_Delay_Timer_7,?,?) XIO(On_Delay_Timer_7.DN) OTE(Station_4A) ,TON(On_Delay_Timer_8,?,?) XIO(On_Delay_Timer_8.DN) OTE(Station_4B) ,TON(On_Delay_Timer_1,?,?) XIO(On_Delay_Timer_1.DN) OTE(Station_5A) ,TON(On_Delay_Timer_2,?,?) XIO(On_Delay_Timer_2.DN) OTE(Station_5B) ,TON(On_Delay_Timer_3,?,?) XIO(On_Delay_Timer_3.DN) OTE(Station_6A) ,TON(On_Delay_Timer_4,?,?) XIO(On_Delay_Timer_4.DN) OTE(Station_6B) ,TON(On_Delay_Timer_5,?,?) XIO(On_Delay_Timer_5.DN) OTE(Station_7A) ,TON(On_Delay_Timer_6,?,?) XIO(On_Delay_Timer_6.DN) OTE(Station_7B) ,TON(On_Delay_Timer_7,?,?) XIO(On_Delay_Timer_7.DN) OTE(Station_8A) ,TON(On_Delay_Timer_8,?,?) XIO(On_Delay_Timer_8.DN) OTE(Station_8B) ];
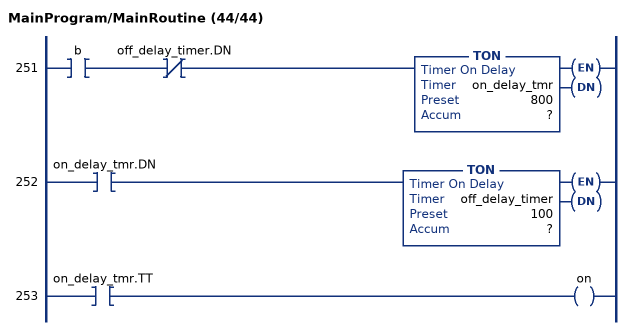
   251: XIC(b)XIO(off_delay_timer.DN)TON(on_delay_tmr,?,?);
   252: XIC(on_delay_tmr.DN)TON(off_delay_timer,?,?);
   253: XIC(on_delay_tmr.TT)OTE(on);
END_ROUTINE
END_PROGRAM
